FUNCTION_BLOCK ExampleCylinderMoveTask EXTENDS TcoCore.TcoTask
VAR_INPUT
	PositionSensor		   : BOOL;
	MaxTimeToReachPosition : TIME := T#10S;
	PositionName		   : STRING(25);
END_VAR
VAR_IN_OUT
	MoveToPositionSignal : BOOL;
	InverseSignal		 : BOOL;	
END_VAR

VAR
	_stringBuilder : TcoCore.StringBuilder;
END_VAR

IF (THIS^.Execute()) THEN
	IF(THIS^.ElapsedTime > MaxTimeToReachPosition) THEN THIS^.Messenger.Warning(_stringBuilder.Clear().Append(PositionName).Append(' sensor not reached yet.').ToString()); END_IF;
	InverseSignal		 := FALSE;
	MoveToPositionSignal := TRUE;
	THIS^.DoneWhen(PositionSensor);	
END_IF

METHOD PUBLIC FB_init : BOOL
VAR_INPUT
	bInitRetains : BOOL; // if TRUE, the retain variables are initialized (warm start / cold start)
	bInCopyCode : BOOL;  // if TRUE, the instance afterwards gets moved into the copy code (online change)
	ParentObject : ITcoObject;
END_VAR
// This is not clear to me... I from time to time the consumer code does not see 'FB_init' of 'TcoObject', that's why overridden here with super call...
//SUPER^.FB_init(bInitRetains, bInCopyCode, ParentObject);
END_METHOD

(*~
	<docu>
		<summary>
			Executes when task is aborted.
		</summary>			
	</docu>	
~*)
METHOD PROTECTED OnAbort
MoveToPositionSignal := FALSE;
END_METHOD

METHOD PROTECTED OnError
END_METHOD

END_FUNCTION_BLOCK

(* stored: Version 1.1.0.1, ProductVersion 3.1.4024.9
   POU ExampleCylinderMoveTask: Id {dff749ca-9903-0426-08d4-2c620927d8bc}, SpecialFunc None
   Method FB_init: Id {c20eb194-2894-0ce3-3f47-dde18deb28e9}
   Method OnAbort: Id {9444377f-e544-0497-18c7-ca5365b44c7c}
   Method OnError: Id {752a0f1c-c464-02a0-035a-76f51036c3fb} *)
